{attribute addProperty BoxType "EP1859-0042-0018"}
{attribute addProperty Id "DI_X01_Pin4AT %I*DI_X01_Pin_E4AEF59E810DI_X01_Pin2AT %I*DI_X01_Pin_E4AEF59E810DI_X02_Pin4AT %I*DI_X02_Pin_E4AEF59E810DI_X02_Pin2AT %I*DI_X02_Pin_E4AEF59E810DI_X03_Pin4AT %I*DI_X03_Pin_E4AEF59E810DI_X03_Pin2AT %I*DI_X03_Pin_E4AEF59E810DI_X04_Pin4AT %I*DI_X04_Pin_E4AEF59E810DI_X04_Pin2AT %I*DI_X04_Pin_E4AEF59E810DO_X05_Pin4AT %Q*DO_X05_Pin_7F374EB0810DO_X05_Pin2AT %Q*DO_X05_Pin_7F374EB0810DO_X06_Pin4AT %Q*DO_X06_Pin_7F374EB0810DO_X06_Pin2AT %Q*DO_X06_Pin_7F374EB0810DO_X07_Pin4AT %Q*DO_X07_Pin_7F374EB0810DO_X07_Pin2AT %Q*DO_X07_Pin_7F374EB0810DO_X08_Pin4AT %Q*DO_X08_Pin_7F374EB0810DO_X08_Pin2AT %Q*DO_X08_Pin_7F374EB0810WcStateAT %I*WcState_98A4DF7520.250InfoDataAT %I*InfoData_192954DE1620"}
{attribute addProperty CRC "651652844"}
{attribute addProperty SizeInBites "146"}
{attribute addProperty SizeInBytes "18.25"}
TYPE EP1859_AFA720D5 :
STRUCT
	{attribute addProperty Name "DI_X01_Pin4"}
	DI_X01_Pin4 : DI_X01_Pin_E4AEF59E;
	{attribute addProperty Name "DI_X01_Pin2"}
	DI_X01_Pin2 : DI_X01_Pin_E4AEF59E;
	{attribute addProperty Name "DI_X02_Pin4"}
	DI_X02_Pin4 : DI_X02_Pin_E4AEF59E;
	{attribute addProperty Name "DI_X02_Pin2"}
	DI_X02_Pin2 : DI_X02_Pin_E4AEF59E;
	{attribute addProperty Name "DI_X03_Pin4"}
	DI_X03_Pin4 : DI_X03_Pin_E4AEF59E;
	{attribute addProperty Name "DI_X03_Pin2"}
	DI_X03_Pin2 : DI_X03_Pin_E4AEF59E;
	{attribute addProperty Name "DI_X04_Pin4"}
	DI_X04_Pin4 : DI_X04_Pin_E4AEF59E;
	{attribute addProperty Name "DI_X04_Pin2"}
	DI_X04_Pin2 : DI_X04_Pin_E4AEF59E;
	{attribute addProperty Name "DO_X05_Pin4"}
	DO_X05_Pin4 : DO_X05_Pin_7F374EB0;
	{attribute addProperty Name "DO_X05_Pin2"}
	DO_X05_Pin2 : DO_X05_Pin_7F374EB0;
	{attribute addProperty Name "DO_X06_Pin4"}
	DO_X06_Pin4 : DO_X06_Pin_7F374EB0;
	{attribute addProperty Name "DO_X06_Pin2"}
	DO_X06_Pin2 : DO_X06_Pin_7F374EB0;
	{attribute addProperty Name "DO_X07_Pin4"}
	DO_X07_Pin4 : DO_X07_Pin_7F374EB0;
	{attribute addProperty Name "DO_X07_Pin2"}
	DO_X07_Pin2 : DO_X07_Pin_7F374EB0;
	{attribute addProperty Name "DO_X08_Pin4"}
	DO_X08_Pin4 : DO_X08_Pin_7F374EB0;
	{attribute addProperty Name "DO_X08_Pin2"}
	DO_X08_Pin2 : DO_X08_Pin_7F374EB0;
	{attribute addProperty Name "WcState"}
	WcState : WcState_98A4DF75;
	{attribute addProperty Name "InfoData"}
	InfoData : InfoData_192954DE;
END_STRUCT
END_TYPE

(* stored: Version 1.2.0.0, ProductVersion 3.1.4024.9
   DUT EP1859_AFA720D5: Id {2d5168e3-e915-4f4b-8f62-fd86902d07c7} *)
